PROGRAM MAIN
VAR
END_VAR

END_PROGRAM

(* stored: Version 1.1.0.1
   POU MAIN: Id {760e1f15-b118-496b-a5df-fbcd2f471756} *)
